// TIA Portal V20 export
TYPE "type_emRelations_em7_sequence"
// stored: Access Published, Namespace Unit1
   STRUCT
      hotPressRight : Struct
         jobs : "LAF_typeJobs";
         sequence : "LAF_typeSequence";
         selectJobStatus { S7_SetPoint := 'True'} : Array[0..10] of "LAF_typeJobStatus";
         "step" : "LER_typeStep";
         jobInterface : Struct
            loadJob2 : "LER_typeJobInterface";
            inspectionJob3 : "LER_typeJobInterface";
            unloadJob4 : "LER_typeJobInterface";
         END_STRUCT;
         homeCheck : Struct
            liftDownPartNoDetect : Bool;
            liftDownPartDetect : Bool;
            liftUp : Bool;
         END_STRUCT;
      END_STRUCT;
   END_STRUCT;
   // // hotPressRight."step".action1[101] : Step[101] : JOB[1] Condition
   // // hotPressRight."step".action1[110] : Step[110] : Servo Press Reference Home Pos
   // // hotPressRight."step".action1[120] : Step[120] : Spare
   // // hotPressRight."step".action1[130] : Step[130] : Spare
   // // hotPressRight."step".action1[140] : Step[140] : Spare
   // // hotPressRight."step".action1[160] : Step[160] : Stage Lift Down
   // // hotPressRight."step".action1[170] : Step[170] : Spare
   // // hotPressRight."step".action1[190] : Step[190] : JOB[1] Step End
   // // hotPressRight."step".action1[201] : Step[201] : JOB[2] Condition
   // // hotPressRight."step".action1[210] : Step[210] : Hot Press Right Loading Request => Transfer PP Left
   // // hotPressRight."step".action1[220] : Step[220] : Spare
   // // hotPressRight."step".action1[230] : Step[230] : Stage Lift Up
   // // hotPressRight."step".action1[240] : Step[240] : Hot Press Right Loading Check => Transfer PP Left
   // // hotPressRight."step".action1[250] : Step[250] : Spare
   // // hotPressRight."step".action1[290] : Step[290] : JOB[2] Step End
   // // hotPressRight."step".action1[301] : Step[301] : JOB[3] Condition
   // // hotPressRight."step".action1[310] : Step[310] : Stage Lift Down
   // // hotPressRight."step".action1[311] : Step[311] : Stage JR Detection Check
   // // hotPressRight."step".action1[320] : Step[320] : Sheet Tension Forward
   // // hotPressRight."step".action1[330] : Step[330] : Hot Press Start
   // // hotPressRight."step".action1[331] : Step[331] : Hot Press Result
   // // hotPressRight."step".action1[380] : Step[380] : Hot Press Home Return
   // // hotPressRight."step".action1[390] : Step[390] : JOB[3] Step End
   // // hotPressRight."step".action1[401] : Step[401] : JOB[4] Condition
   // // hotPressRight."step".action1[410] : Step[410] : Spare
   // // hotPressRight."step".action1[420] : Step[420] : Stage Lift Up
   // // hotPressRight."step".action1[430] : Step[430] : Hot Press Right Unloading Request => Transfer PP Left
   // // hotPressRight."step".action1[431] : Step[431] : Hot Press Right Unloading Check => Transfer PP Left
   // // hotPressRight."step".action1[480] : Step[480] : Stage Lift Down
   // // hotPressRight."step".action1[481] : Step[481] : Spare
   // // hotPressRight."step".action1[490] : Step[490] : JOB[4] Step End
   // // hotPressRight."step".transition1[101] : Step[101] : JOB[1] Condition
   // // hotPressRight."step".transition1[110] : Step[110] : Servo Press Reference Home Pos
   // // hotPressRight."step".transition1[120] : Step[120] : Spare
   // // hotPressRight."step".transition1[130] : Step[130] : Spare
   // // hotPressRight."step".transition1[140] : Step[140] : Spare
   // // hotPressRight."step".transition1[160] : Step[160] : Stage Lift Down
   // // hotPressRight."step".transition1[170] : Step[170] : Spare
   // // hotPressRight."step".transition1[190] : Step[190] : JOB[1] Step End
   // // hotPressRight."step".transition1[201] : Step[201] : JOB[2] Condition
   // // hotPressRight."step".transition1[210] : Step[210] : Hot Press Right Loading Request => Transfer PP Left
   // // hotPressRight."step".transition1[220] : Step[220] : Spare
   // // hotPressRight."step".transition1[230] : Step[230] : Stage Lift Up
   // // hotPressRight."step".transition1[240] : Step[240] : Hot Press Right Loading Check => Transfer PP Left
   // // hotPressRight."step".transition1[250] : Step[250] : Spare
   // // hotPressRight."step".transition1[290] : Step[290] : JOB[2] Step End
   // // hotPressRight."step".transition1[301] : Step[301] : JOB[3] Condition
   // // hotPressRight."step".transition1[310] : Step[310] : Stage Lift Down
   // // hotPressRight."step".transition1[311] : Step[311] : Stage JR Detection Check
   // // hotPressRight."step".transition1[320] : Step[320] : Sheet Tension Forward
   // // hotPressRight."step".transition1[330] : Step[330] : Hot Press Start
   // // hotPressRight."step".transition1[331] : Step[331] : Hot Press Result
   // // hotPressRight."step".transition1[380] : Step[380] : Hot Press Home Return
   // // hotPressRight."step".transition1[390] : Step[390] : JOB[3] Step End
   // // hotPressRight."step".transition1[401] : Step[401] : JOB[4] Condition
   // // hotPressRight."step".transition1[410] : Step[410] : Spare
   // // hotPressRight."step".transition1[420] : Step[420] : Stage Lift Up
   // // hotPressRight."step".transition1[430] : Step[430] : Hot Press Right Unloading Request => Transfer PP Left
   // // hotPressRight."step".transition1[431] : Step[431] : Hot Press Right Unloading Check => Transfer PP Left
   // // hotPressRight."step".transition1[480] : Step[480] : Stage Lift Down
   // // hotPressRight."step".transition1[481] : Step[481] : Spare
   // // hotPressRight."step".transition1[490] : Step[490] : JOB[4] Step End
END_TYPE
